Yaskawa INFORM job: OK_R2_O55(0,90)_AWOK.JBI

/JOB
//NAME OK_R2_O55(0,90)_AWOK
///FOLDERNAME X4
//POS
///NPOS 380,380,380,6,0,0
///TOOL 0
///POSTYPE PULSE
///PULSE
C00000=-116137,-64682,-98842,-22895,83957,21003
C00001=-118970,-58791,-94528,-21719,83626,20151
C00002=-128709,-21936,-78165,-7667,99802,18846
C00003=-128709,-23747,-77378,-7629,98400,18933
C00004=-129436,-40962,-90086,-7600,97096,18720
C00005=-119723,-61472,-87397,-21694,78070,20911
C00006=-121447,-61479,-87400,-20976,77655,20398
C00007=-122276,-61450,-87381,-20627,77465,20150
C00008=-121447,-61479,-87400,-20976,77655,20398
C00009=-119962,-55971,-84809,-21515,79163,20631
C00010=-119972,-52981,-83428,-21469,79803,20512
C00011=-119962,-55971,-84809,-21515,79163,20631
C00012=-118927,-58061,-86775,-21934,79541,20910
C00013=-116191,-63318,-91619,-23033,80483,21654
C00014=-116206,-56841,-96943,-22807,86586,20479
C00015=-116389,-60342,-95375,-22789,83985,20915
C00016=-116893,-39967,-83874,-22518,87009,20183
C00017=-125017,-21387,-77981,-10790,100136,18660
C00018=-125017,-23744,-76950,-10720,98321,18819
C00019=-116787,-42854,-87540,-22390,92348,19284
C00020=-121082,-61460,-87305,-21133,77696,20515
C00021=-121082,-61460,-87305,-21133,77696,20515
C00022=-122532,-61410,-87275,-20524,77362,20082
C00023=-121082,-61460,-87305,-21133,77696,20515
C00024=-120060,-56933,-85154,-21492,78877,20650
C00025=-120072,-53043,-83376,-21432,79719,20494
C00026=-120060,-56933,-85154,-21492,78877,20650
C00027=-119021,-59046,-87123,-21913,79246,20933
C00028=-116273,-64366,-91974,-23018,80167,21688
C00029=-116287,-57977,-97359,-22777,86263,20515
C00030=-114907,-63183,-96670,-23411,83739,21445
C00031=-115618,-41571,-84692,-23045,87010,20581
C00032=-116115,-23132,-74965,-22736,98208,18438
C00033=-116115,-24314,-74310,-22669,97276,18619
C00034=-115586,-41490,-86592,-22768,96199,18989
C00035=-121083,-61695,-87340,-21139,77603,20531
C00036=-121083,-61695,-87340,-21139,77603,20531
C00037=-122529,-61648,-87311,-20532,77268,20097
C00038=-121083,-61695,-87340,-21139,77603,20531
C00039=-120059,-57166,-85192,-21498,78788,20666
C00040=-120072,-53268,-83414,-21438,79633,20510
C00041=-120059,-57166,-85192,-21498,78788,20666
C00042=-119019,-59284,-87162,-21920,79155,20951
C00043=-116268,-64618,-92014,-23026,80071,21708
C00044=-116282,-58266,-97419,-22781,86162,20535
C00045=-116234,-65654,-98856,-22870,83480,21063
C00046=-117001,-30938,-83151,-22477,97538,18275
C00047=-117162,-27122,-76676,-22301,95626,18585
C00048=-117162,-28033,-76136,-22264,94882,18725
C00049=-116792,-43513,-86705,-22330,93619,19076
C00050=-121083,-61930,-87375,-21146,77510,20548
C00051=-121083,-61930,-87375,-21146,77510,20548
C00052=-122667,-61875,-87342,-20480,77145,20073
C00053=-121083,-61930,-87375,-21146,77510,20548
C00054=-120059,-57398,-85231,-21504,78698,20682
C00055=-120071,-53441,-83423,-21444,79555,20523
C00056=-120059,-57398,-85231,-21504,78698,20682
C00057=-119017,-59522,-87201,-21927,79064,20968
C00058=-116262,-64869,-92054,-23034,79975,21729
C00059=-116277,-58554,-97479,-22785,86060,20556
C00060=-116228,-66833,-98171,-22911,82531,21247
C00061=-117126,-25406,-79498,-22565,100598,17692
C00062=-117248,-21815,-74608,-22429,99491,17867
C00063=-117248,-22912,-74026,-22358,98638,18029
C00064=-116836,-40210,-86441,-22404,97572,18358
C00065=-121084,-62164,-87410,-21153,77417,20564
C00066=-121084,-62164,-87410,-21153,77417,20564
C00067=-122661,-62109,-87376,-20489,77054,20090
C00068=-121084,-62164,-87410,-21153,77417,20564
C00069=-120058,-57630,-85269,-21511,78609,20699
C00070=-120070,-53643,-83448,-21448,79472,20539
C00071=-120058,-57630,-85269,-21511,78609,20699
C00072=-119015,-59759,-87239,-21934,78973,20985
C00073=-116257,-65120,-92093,-23043,79880,21749
C00074=-116279,-54556,-99745,-22770,89251,19950
C00075=-114774,-111312,-123896,-23941,76439,22953
C00076=-117925,-58719,-95873,-21124,87917,23523
C00077=-103186,-10021,-58133,-44610,101398,29068
C00078=-123420,-23872,-71025,-15792,95845,28310
C00079=-125311,-21429,-67110,-15147,94424,27919
C00080=-120634,-65913,-76142,-32119,72760,24735
C00081=-119236,-64284,-74350,-32649,73056,25211
C00082=-125319,-21707,-67309,-15144,94403,27919
C00083=-125467,-27325,-70565,-15073,93526,27983
C00084=-125604,-31584,-72851,-15014,92748,28038
C00085=-123522,-33905,-76479,-15704,94095,28507
C00086=-123564,-36325,-78032,-15683,93810,28531
C00087=-119101,-30822,-74067,-21861,99204,35368
C00088=-119596,-32319,-75056,-21718,98940,35258
C00089=-119766,-30799,-71819,-21590,97773,35415
C00090=-121301,-29842,-70621,-21174,97189,35027
C00091=-119239,-57603,-89587,-23561,101073,42379
C00092=-120637,-57975,-90978,-23357,101328,41854
C00093=-121301,-29842,-70621,-21174,97189,35027
C00094=-121414,-33462,-72174,-21093,96316,35147
C00095=-121364,-37608,-74051,-21057,95413,35322
C00096=-118165,-36043,-78158,-22099,99263,35661
C00097=-118125,-31017,-84138,-22729,105083,34553
C00098=-120714,-60708,-105430,-21771,102512,34247
C00099=-95484,-136154,-93871,-55672,51405,46786
C00100=-114713,-99798,-82990,-41844,49051,35906
C00101=-120637,-59624,-88700,-22681,87253,37649
C00102=-119238,-59498,-87405,-23139,86931,38179
C00103=-114711,-99839,-83005,-41852,49043,35911
C00104=-114545,-102590,-83009,-42762,48062,36535
C00105=-114219,-107980,-82478,-44894,45954,37960
C00106=-111898,-109767,-89828,-42010,51787,36738
C00107=-111805,-126727,-95079,-45212,47795,38991
C00108=-66535,-95601,-84684,-52007,78764,46851
C00109=-75218,-92548,-82480,-50699,74029,44853
C00110=-81141,-84946,-78957,-49165,71925,42856
C00111=-123268,-63523,-79231,-37570,63516,21441
C00112=-124736,-66195,-80529,-37014,62443,21190
C00113=-81122,-84998,-78949,-49177,71915,42872
C00114=-79718,-88775,-78946,-49929,71393,43910
C00115=-78361,-92195,-78675,-50655,70883,44930
C00116=-68284,-113231,-96700,-52052,76723,47086
C00117=-66672,-117056,-107174,-51639,80473,45806
C00118=-77691,-86619,-95818,-48386,80174,40315
C00119=-95685,-48808,-84743,-25370,87231,35181
C00120=-95685,-48808,-84743,-25370,87231,35181
C00121=-101056,-45173,-78089,-23427,83774,34106
C00122=-102119,-43985,-76293,-23044,83049,33893
C00123=-122027,-64752,-74386,33128,72903,-25284
C00124=-120634,-66395,-76191,32602,72601,-24811
C00125=-102106,-44094,-76359,-23049,83038,33899
C00126=-101400,-49999,-79288,-23366,82078,34324
C00127=-100787,-55009,-81515,-23654,81130,34721
C00128=-99386,-53621,-81963,-24126,82412,34943
C00129=-94381,-41540,-79397,-29257,97383,37091
C00130=-94381,-42754,-78179,-29152,96177,37399
C00131=-94595,-42729,-76833,-29043,95394,37523
C00132=-96175,-42441,-75420,-28594,94264,37251
C00133=-120637,-58450,-91149,23792,101183,-41860
C00134=-122028,-58068,-89746,23994,100932,-42385
C00135=-96165,-42504,-75459,-28596,94259,37256
C00136=-95794,-45065,-76561,-28658,93810,37497
C00137=-95105,-50085,-78357,-28765,92724,38011
C00138=-93482,-48166,-78689,-29220,94287,38194
C00139=-91547,-49523,-92929,-30449,101938,36857
C00140=-111094,-45126,-96422,5689,101572,-12606
C00141=-121972,-50267,-96226,12386,99274,-20777
C00142=-120632,-57742,-90169,23117,88968,-37302
C00143=-120632,-59368,-88362,23119,87170,-37649
C00144=-119891,-47131,-80888,22873,88542,-37139
C00145=-122028,-59922,-87589,23577,86831,-38184
C00146=-120637,-60056,-88897,23120,87149,-37655
C00147=-119891,-47131,-80888,22873,88542,-37139
C00148=-120005,-53355,-83923,22914,87335,-37405
C00149=-119935,-58609,-86237,22903,86131,-37610
C00150=-123325,-57174,-87874,23990,88618,-38260
C00151=-124456,-73122,-93330,24403,84490,-39484
C00152=-120301,-77332,-95283,21145,80945,-36635
C00153=-117644,-75175,-92925,20247,79987,-35884
C00154=-120632,-66782,-80600,39533,64000,-22464
C00155=-122028,-63953,-79218,40005,65086,-22660
C00156=-117642,-75287,-92977,20248,79962,-35887
C00157=-117577,-78550,-93986,20282,78953,-36035
C00158=-117430,-84106,-95504,20358,77113,-36296
C00159=-121605,-82442,-100182,21565,81626,-36962
C00160=-121605,-75018,-107752,21416,89537,-35553
C00161=-98045,-149302,-129631,14244,61097,-31502
C00162=-124074,-173592,-119291,35973,43889,-32820
C00163=-132864,-143257,-102711,42749,53298,-34446
C00164=-130839,-124766,-99786,38797,58274,-31089
C00165=-123631,-118072,-96989,34608,55995,-27816
C00166=-123631,-118072,-96989,34608,55995,-27816
C00167=-123717,-121009,-96897,35249,54734,-28334
C00168=-124024,-127264,-96467,36865,52023,-29582
C00169=-126943,-131602,-98873,38274,52691,-30822
C00170=-128360,-153372,-105295,42598,47752,-34029
C00171=-79453,-131856,-104511,4352,44365,-9914
C00172=-78436,-115658,-92400,1620,36378,-6800
C00173=-77806,-111855,-90740,987,37302,-6435
C00174=-120634,-65728,-76133,-32106,72837,24713
C00175=-119238,-64103,-74341,-32635,73130,25188
C00176=-77806,-111855,-90740,987,37302,-6435
C00177=-76429,-114788,-90587,-338,35694,-5673
C00178=-73763,-118985,-89653,-3164,33028,-4038
C00179=-66359,-139525,-96150,-13144,27249,1592
C00180=-66359,-164100,-123806,-11486,31545,742
C00181=-70302,-83518,-108233,-11696,76370,-6987
C00182=-79254,-60990,-87055,-7574,73946,-9698
C00183=-79142,-57343,-85120,-7603,74633,-9705
C00184=-85366,-48204,-80333,1212,78686,-14938
C00185=-119241,-57353,-89541,-23570,101165,42360
C00186=-120637,-57719,-90930,-23367,101422,41835
C00187=-85366,-48204,-80333,1212,78686,-14938
C00188=-84294,-52923,-82551,739,77615,-14611
C00189=-82864,-58973,-85150,105,76099,-14163
C00190=-83777,-59837,-86544,514,76516,-14454
C00191=-81015,-69582,-89979,-723,73625,-13560
C00192=-84711,-68031,-88236,4430,73597,-17336
C00193=-120637,-59381,-88659,-22680,87345,37632
C00194=-119240,-59261,-87366,-23138,87022,38161
C00195=-84711,-68031,-88236,4430,73597,-17336
C00196=-83691,-72246,-89459,4003,72137,-17046
C00197=-83032,-75359,-90390,3727,71082,-16859
C00198=-84024,-76098,-91808,4166,71620,-17177
C00199=-84024,-66051,-103222,3998,83778,-16777
C00200=-65662,-31425,-83606,-4017,89486,-11563
C00201=-68948,-27521,-69076,-2600,82448,-12318
C00202=-64522,-19418,-61513,-8839,82863,-8015
C00203=-119239,-63197,-79148,-39462,65333,22543
C00204=-120631,-66018,-80525,-38983,64255,22343
C00205=-64522,-19418,-61513,-8839,82863,-8015
C00206=-63064,-23118,-63668,-9464,82443,-7541
C00207=-61424,-27145,-65833,-10171,81894,-6997
C00208=-62353,-28195,-68036,-9762,82596,-7338
C00209=-64122,-27053,-68918,-6328,85296,-12363
C00210=-62252,-32477,-70641,-7099,83718,-11715
C00211=-63845,-35903,-70208,-3997,79095,-11410
C00212=-122025,-64571,-74378,33114,72977,-25261
C00213=-120634,-66211,-76182,32588,72677,-24788
C00214=-63845,-35903,-70208,-3997,79095,-11410
C00215=-62658,-39020,-71374,-4529,78269,-11011
C00216=-61692,-41451,-72189,-4965,77573,-10680
C00217=-64197,-44187,-78529,-3833,79939,-11548
C00218=-64197,-33780,-85787,-3792,89732,-11844
C00219=-44689,-70929,-106175,-12114,84890,-5931
C00220=-33806,-93502,-88404,-27904,59082,13170
C00221=-58177,-75417,-81541,-6000,56276,1441
C00222=-58430,-67739,-76898,-5771,57341,1282
C00223=-120637,-58195,-91102,23802,101277,-41841
C00224=-122027,-57818,-89700,24003,101023,-42366
C00225=-58430,-67739,-76898,-5771,57341,1282
C00226=-58984,-71347,-77159,-3299,55423,-230
C00227=-57144,-74611,-77050,-4586,53771,576
C00228=-50982,-91677,-90407,-7950,54776,1850
C00229=-50982,-85567,-109418,-6960,69497,875
C00230=-54812,-62849,-98997,-4717,74482,-585
C00231=-50289,-1036,-61538,-16344,96039,-3895
C00232=-52048,7040,-42367,-12868,86243,-4159
C00233=-56434,8881,-38977,-5883,83428,-8939
C00234=-122026,-59684,-87550,23576,86921,-38166
C00235=-120637,-59813,-88856,23120,87241,-37637
C00236=-56434,8881,-38977,-5883,83428,-8939
C00237=-55375,6495,-40648,-6339,83302,-8616
C00238=-53560,2556,-43263,-7119,83025,-8054
C00239=-54077,1434,-44695,-6896,83288,-8224
C00240=-50741,-4405,-49866,-7836,84192,-7156
C00241=-51041,-4740,-48575,-7721,83208,-7185
C00242=-51232,-2335,-46154,-7645,82940,-7226
C00243=-120632,-66582,-80584,39505,64073,-22434
C00244=-122026,-63754,-79201,39978,65156,-22630
C00245=-51232,-2335,-46154,-7645,82940,-7226
C00246=-50099,-4713,-47267,-8126,82505,-6854
C00247=-49243,-6461,-48043,-8490,82167,-6570
C00248=-50339,-8396,-52000,-8013,83495,-6993
C00249=-50339,-276,-57860,-7996,91201,-7484
C00250=-32565,-26345,-77616,-15225,92076,-2559
C00251=-32565,-33689,-72287,-15210,85259,-1719
C00252=-38687,-36831,-55238,-24407,59977,6052
C00253=-39203,-33265,-53072,-24000,60287,5772
C00254=-120634,-65542,-76123,-32092,72913,24690
C00255=-119239,-63920,-74332,-32621,73204,25165
C00256=-39203,-33265,-53072,-24000,60287,5772
C00257=-37714,-35062,-52939,-25083,59795,6495
C00258=-35590,-37744,-52712,-26656,59062,7564
C00259=-26545,-57404,-66697,-31827,60841,10944
C00260=-20629,-19497,-42558,-33469,66981,11514
C00261=-27693,-14289,-39743,-29849,65249,9144
C00262=-34880,-670,-29098,-19183,60278,2827
C00263=-35092,1454,-27069,-19082,60082,2779
C00264=-119242,-57104,-89496,-23579,101256,42341
C00265=-120637,-57464,-90882,-23377,101516,41817
C00266=-35092,1454,-27069,-19082,60082,2779
C00267=-33603,-474,-27156,-20166,59534,3463
C00268=-32057,-2336,-26931,-21326,58881,4207
C00269=-32408,-6201,-31843,-20897,59764,3889
C00270=-24820,-12827,-37041,-25332,61618,6510
C00271=-24820,-941,-54339,-22867,76995,3228
C00272=-42185,7615,-42322,-13268,70874,-1244
C00273=-42932,41857,-5727,-16679,81128,-4248
C00274=-120637,-59139,-88618,-22679,87437,37614
C00275=-119242,-59024,-87327,-23137,87112,38143
C00276=-42935,41623,-5955,-16677,81147,-4251
C00277=-41455,39000,-8178,-17284,81445,-3818
C00278=-40207,36838,-9888,-17795,81632,-3440
C00279=-40859,34117,-14035,-17490,82609,-3791
C00280=-37683,30675,-15388,-18805,82352,-2733
C00281=-37683,30675,-15388,-18805,82352,-2733
C00282=-37615,32337,-12840,-18862,81691,-2611
C00283=-119240,-62997,-79129,-39436,65404,22513
C00284=-120631,-65817,-80509,-38956,64328,22314
C00285=-37615,32337,-12840,-18862,81691,-2611
C00286=-36831,30953,-13603,-19182,81626,-2349
C00287=-35920,29533,-14307,-19552,81540,-2037
C00288=-36765,31666,-24197,-19069,88162,-3353
C00289=-80819,-21628,-74687,-2656,88110,49135
C00290=-52229,28768,-25499,-44312,108635,44591
C00291=-56025,35229,-16083,-42906,105184,44544
C00292=-61493,29391,-19794,-36258,100135,45607
C00293=-62872,29148,-18454,-35815,98844,45518
C00294=-122023,-64389,-74369,33100,73050,-25238
C00295=-120634,-66025,-76173,32574,72753,-24766
C00296=-62615,28475,-19058,-35877,98962,45577
C00297=-61224,24817,-22216,-36208,99536,45909
C00298=-60367,22322,-24134,-36395,99777,46151
C00299=-59915,24005,-23707,-36577,100438,46097
C00300=-56946,22626,-23553,-38393,103359,48615
C00301=-57829,21509,-23426,-38110,102492,48585
C00302=-120637,-57938,-91054,23812,101371,-41822
C00303=-122025,-57567,-89654,24013,101115,-42346
C00304=-57829,21509,-23426,-38110,102492,48585
C00305=-56932,18945,-24988,-38222,102566,48914
C00306=-56106,16994,-26094,-38319,102642,49215
C00307=-54980,21729,-25214,-38868,104590,48938
C00308=-54302,30399,-28737,-40542,110020,47060
C00309=-40953,8747,-49252,-43839,116433,49649
C00310=-43706,2890,-35678,-39962,106692,52751
C00311=-46557,4892,-23316,-53006,96166,51821
C00312=-122025,-59445,-87511,23574,87012,-38148
C00313=-120637,-59568,-88815,23119,87334,-37619
C00314=-46557,4892,-23316,-53006,96166,51821
C00315=-45252,2504,-23846,-53101,96327,52417
C00316=-43850,228,-24056,-53173,96460,53085
C00317=-40014,1377,-25111,-53867,99354,53399
C00318=-32910,-4730,-38816,-56031,106441,52743
C00319=-47083,-38904,-60179,-52956,95987,51646
C00320=-56245,-29117,-51675,-51253,90891,49843
C00321=-59207,-29685,-49787,-50620,88366,49736
C00322=-120632,-66381,-80568,39477,64146,-22405
C00323=-122024,-63554,-79183,39951,65226,-22600
C00324=-59207,-29685,-49787,-50620,88366,49736
C00325=-57910,-32588,-50321,-50873,88309,50423
C00326=-56386,-35626,-50587,-51149,88234,51241
C00327=-48005,-36349,-53024,-52514,93554,52587
C00328=-45972,-31923,-70966,-54898,102784,48011
C00329=-62213,-2026,-48801,-50558,95689,44317
C00330=-71635,-10765,-49348,-38257,85995,47822
C00331=-73562,-12108,-48704,-37621,84358,47652
C00332=-120634,-65355,-76113,-32078,72990,24668
C00333=-119241,-63738,-74323,-32607,73278,25142
C00334=-73562,-12108,-48704,-37621,84358,47652
C00335=-72319,-16326,-51343,-38077,84425,48112
C00336=-71460,-18971,-52889,-38389,84454,48442
C00337=-69249,-19212,-54152,-39109,85879,48797
C00338=-68409,7690,-37813,-43127,101148,56069
C00339=-66304,155,-40606,-43261,100476,57243
C00340=-68124,-581,-39889,-42746,99066,57077
C00341=-119244,-56851,-89448,-23589,101349,42322
C00342=-120637,-57205,-90833,-23387,101611,41798
C00343=-68124,-581,-39889,-42746,99066,57077
C00344=-67510,-2508,-40929,-42832,99077,57331
C00345=-66648,-5140,-42298,-42942,99083,57691
C00346=-65956,-2564,-42142,-43266,100302,57463
C00347=-64160,8326,-48156,-45635,107840,54777
C00348=-82891,-1763,-56772,-40060,100398,50695
C00349=-87672,-9018,-50191,-37820,92424,51832
C00350=-88713,-8713,-49183,-37485,91645,51714
C00351=-120636,-58892,-88576,-22679,87531,37597
C00352=-119243,-58782,-87287,-23135,87203,38125
C00353=-88713,-8713,-49183,-37485,91645,51714
C00354=-87862,-13103,-52108,-37724,91615,52052
C00355=-87153,-16713,-54260,-37916,91475,52374
C00356=-86564,-15302,-54870,-38138,92586,52206
C00357=-81758,-3749,-44861,-44343,103015,58118
C00358=-82859,-4851,-44447,-43969,101921,58133
C00359=-83726,-5948,-44324,-43688,101062,58138
C00360=-119242,-62796,-79110,-39409,65475,22484
C00361=-120631,-65615,-80491,-38929,64402,22285
C00362=-83726,-5948,-44324,-43688,101062,58138
C00363=-83153,-8645,-45822,-43726,100977,58421
C00364=-82498,-11692,-47360,-43751,100817,58774
C00365=-79946,-9385,-47908,-44504,103092,58867
C00366=-79946,982,-56626,-47228,110687,55169
C00367=-67961,-35581,-83522,-49317,114444,58500
C00368=-66559,-58522,-69059,-49468,91172,57867
C00369=-76672,-55097,-64494,-49467,77742,54734
C00370=-122022,-64207,-74360,33086,73124,-25215
C00371=-120634,-65839,-76164,32560,72829,-24743
C00372=-76672,-55097,-64494,-49467,77742,54734
C00373=-75645,-58080,-64974,-49897,77474,55402
C00374=-74048,-62341,-65191,-50569,76997,56494
C00375=-72098,-59878,-66217,-50707,79300,56246
C00376=-48660,-78559,-75441,-54167,90144,62579
C00377=-24519,-71348,-75508,-48873,52324,28946
C00378=-2117,-60454,-47312,-54295,7475,4900
C00379=-2158,-60407,-47353,-53850,7490,4702
BC00000=362177,692409,1075175
BC00001=362177,692409,1075175
BC00002=362177,692409,1075175
BC00003=362177,692409,1075175
BC00004=362177,692409,1075175
BC00005=362177,692409,1075175
BC00006=362177,692409,1075175
BC00007=362177,692409,1075175
BC00008=362177,692409,1075175
BC00009=362177,692409,1075175
BC00010=362177,692409,1075175
BC00011=362177,692409,1075175
BC00012=362177,692409,1075175
BC00013=362177,692409,1075175
BC00014=362177,692409,1075175
BC00015=314570,692300,1075175
BC00016=314570,692300,1075175
BC00017=314571,692301,1075171
BC00018=314571,692301,1075171
BC00019=314570,692300,1075175
BC00020=314570,692300,1075175
BC00021=314570,692300,1075175
BC00022=314570,692300,1075175
BC00023=314570,692300,1075175
BC00024=314570,692300,1075175
BC00025=314570,692300,1075175
BC00026=314570,692300,1075175
BC00027=314570,692300,1075175
BC00028=314570,692300,1075175
BC00029=314570,692300,1075175
BC00030=266548,692394,1075175
BC00031=266548,692394,1075175
BC00032=266548,692394,1075175
BC00033=266548,692394,1075175
BC00034=266548,692394,1075175
BC00035=266548,692394,1075175
BC00036=266548,692394,1075175
BC00037=266548,692394,1075175
BC00038=266548,692394,1075175
BC00039=266548,692394,1075175
BC00040=266548,692394,1075175
BC00041=266548,692394,1075175
BC00042=266548,692394,1075175
BC00043=266548,692394,1075175
BC00044=266548,692394,1075175
BC00045=218526,692488,1075175
BC00046=218526,692488,1075175
BC00047=218526,692488,1075175
BC00048=218526,692488,1075175
BC00049=218526,692488,1075175
BC00050=218526,692488,1075175
BC00051=218526,692488,1075175
BC00052=218526,692488,1075175
BC00053=218526,692488,1075175
BC00054=218526,692488,1075175
BC00055=218526,692488,1075175
BC00056=218526,692488,1075175
BC00057=218526,692488,1075175
BC00058=218526,692488,1075175
BC00059=218526,692488,1075175
BC00060=170743,692582,1075175
BC00061=170743,692582,1075175
BC00062=170743,692582,1075175
BC00063=170743,692582,1075175
BC00064=170743,692582,1075175
BC00065=170743,692582,1075175
BC00066=170743,692582,1075175
BC00067=170743,692582,1075175
BC00068=170743,692582,1075175
BC00069=170743,692582,1075175
BC00070=170743,692582,1075175
BC00071=170743,692582,1075175
BC00072=170743,692582,1075175
BC00073=170743,692582,1075175
BC00074=170743,692582,1075175
BC00075=170743,673726,1075175
BC00076=170861,676324,1075173
BC00077=170861,676324,1075173
BC00078=171122,682063,1075169
BC00079=171122,682063,1075169
BC00080=184393,664970,1075175
BC00081=184393,664970,1075175
BC00082=171122,682063,1075169
BC00083=171122,682063,1075169
BC00084=171122,682063,1075169
BC00085=171122,682063,1075169
BC00086=171122,682063,1075169
BC00087=171122,682063,1075169
BC00088=171122,682063,1075169
BC00089=171122,682063,1075169
BC00090=171122,682063,1075169
BC00091=173178,720507,1075175
BC00092=173178,720507,1075175
BC00093=171122,682063,1075169
BC00094=171122,682063,1075169
BC00095=171122,682063,1075169
BC00096=171122,682063,1075169
BC00097=171122,682063,1075169
BC00098=171122,682063,1075169
BC00099=171122,682063,1075169
BC00100=171122,682063,1075169
BC00101=173051,704467,1075175
BC00102=173051,704467,1075175
BC00103=171122,682063,1075169
BC00104=171122,682063,1075169
BC00105=171122,682063,1075169
BC00106=171498,685555,1075169
BC00107=171498,685555,1075169
BC00108=171498,685555,1075169
BC00109=171498,685555,1075169
BC00110=171498,685555,1075169
BC00111=196106,690466,1075175
BC00112=196106,690466,1075175
BC00113=171498,685555,1075169
BC00114=171498,685555,1075169
BC00115=171498,685555,1075169
BC00116=171498,685555,1075169
BC00117=171498,685555,1075169
BC00118=171498,685555,1075169
BC00119=171731,685521,1075169
BC00120=171731,685521,1075169
BC00121=171731,685521,1075169
BC00122=171731,685521,1075169
BC00123=58729,665797,1075175
BC00124=58729,665797,1075175
BC00125=171731,685521,1075169
BC00126=171731,685521,1075169
BC00127=171731,685521,1075169
BC00128=171731,685521,1075169
BC00129=171731,685521,1075169
BC00130=171731,685521,1075169
BC00131=171731,685521,1075169
BC00132=171731,685521,1075169
BC00133=70497,721413,1075175
BC00134=70497,721413,1075175
BC00135=171731,685521,1075169
BC00136=171731,685521,1075169
BC00137=171731,685521,1075169
BC00138=171731,685521,1075169
BC00139=171731,685521,1075169
BC00140=98396,696294,1075173
BC00141=90128,697509,1075173
BC00142=62613,701551,1075175
BC00143=68182,704259,1075175
BC00144=69760,705026,1075175
BC00145=70409,705342,1075175
BC00146=70409,705342,1075175
BC00147=69760,705026,1075175
BC00148=69760,705026,1075175
BC00149=69760,705026,1075175
BC00150=69760,705026,1075175
BC00151=69760,705026,1075175
BC00152=69760,705026,1075175
BC00153=69760,705026,1075175
BC00154=53891,691077,1075175
BC00155=53891,691077,1075175
BC00156=69760,705026,1075175
BC00157=69760,705026,1075175
BC00158=69760,705026,1075175
BC00159=69760,705026,1075175
BC00160=69760,705026,1075175
BC00161=69760,705026,1075175
BC00162=69760,705026,1075175
BC00163=69760,705026,1075175
BC00164=69760,705026,1075175
BC00165=69760,705026,1075175
BC00166=69760,705026,1075175
BC00167=69760,705026,1075175
BC00168=69760,705026,1075175
BC00169=69760,705026,1075175
BC00170=69760,705026,1075175
BC00171=69760,705026,1075175
BC00172=69760,705026,1075175
BC00173=69760,705026,1075175
BC00174=232176,664876,1075175
BC00175=232176,664876,1075175
BC00176=69760,705026,1075175
BC00177=69760,705026,1075175
BC00178=69760,705026,1075171
BC00179=69760,705026,1075171
BC00180=69760,705026,1075171
BC00181=69760,705026,1075171
BC00182=69760,705026,1075171
BC00183=69760,705026,1075171
BC00184=69760,705026,1075171
BC00185=220961,720413,1075175
BC00186=220961,720413,1075175
BC00187=69760,705026,1075171
BC00188=69760,705026,1075171
BC00189=69760,705026,1075171
BC00190=69760,705026,1075171
BC00191=69760,705026,1075171
BC00192=69760,705026,1075171
BC00193=220834,704373,1075175
BC00194=220834,704373,1075175
BC00195=69760,705026,1075171
BC00196=69760,705026,1075171
BC00197=69760,705026,1075171
BC00198=69760,705026,1075171
BC00199=69760,705026,1075171
BC00200=69760,705026,1075171
BC00201=69760,705026,1075171
BC00202=69760,705026,1075171
BC00203=236979,690198,1075175
BC00204=236979,690198,1075175
BC00205=69760,705026,1075171
BC00206=69760,705026,1075171
BC00207=69760,705026,1075171
BC00208=69760,705026,1075171
BC00209=69760,705026,1075171
BC00210=69760,705026,1075171
BC00211=69760,705026,1075171
BC00212=106512,665703,1075175
BC00213=106512,665703,1075175
BC00214=69760,705026,1075171
BC00215=69760,705026,1075171
BC00216=69760,705026,1075171
BC00217=69760,705026,1075171
BC00218=69760,705026,1075171
BC00219=69760,705026,1075171
BC00220=69760,705026,1075171
BC00221=70001,705106,1075155
BC00222=70001,705106,1075155
BC00223=118281,721319,1075175
BC00224=118281,721319,1075175
BC00225=70001,705106,1075155
BC00226=70001,705106,1075161
BC00227=70001,705106,1075165
BC00228=72274,705262,1075165
BC00229=72274,705262,1075165
BC00230=72274,705262,1075165
BC00231=72274,705262,1075165
BC00232=72274,705262,1075165
BC00233=72274,705262,1075165
BC00234=118193,705249,1075175
BC00235=118193,705249,1075175
BC00236=72274,705262,1075165
BC00237=72274,705262,1075165
BC00238=72274,705262,1075165
BC00239=72274,705262,1075165
BC00240=72274,705262,1075165
BC00241=72274,705262,1075165
BC00242=72274,705262,1075165
BC00243=101675,690983,1075175
BC00244=101675,690983,1075175
BC00245=72274,705262,1075165
BC00246=72274,705262,1075165
BC00247=72274,705262,1075165
BC00248=72274,705262,1075165
BC00249=72274,705262,1075165
BC00250=72274,705262,1075165
BC00251=72274,705262,1075165
BC00252=72274,705262,1075165
BC00253=72274,705262,1075165
BC00254=280198,664783,1075175
BC00255=280198,664783,1075175
BC00256=72274,705262,1075165
BC00257=72274,705262,1075165
BC00258=72274,705262,1075165
BC00259=72274,705262,1075165
BC00260=72274,705262,1075165
BC00261=72274,705262,1075165
BC00262=72274,705262,1075165
BC00263=72274,705262,1075165
BC00264=268505,720320,1075175
BC00265=268505,720320,1075175
BC00266=72274,705262,1075165
BC00267=72274,705262,1075165
BC00268=72274,705262,1075165
BC00269=72274,705262,1075165
BC00270=72274,705262,1075165
BC00271=72274,705262,1075165
BC00272=72274,705262,1075165
BC00273=72274,705261,1075162
BC00274=268378,704280,1075175
BC00275=268378,704280,1075175
BC00276=72274,705261,1075162
BC00277=72274,705262,1075165
BC00278=72274,705262,1075165
BC00279=72274,705262,1075165
BC00280=72274,705262,1075165
BC00281=72274,705262,1075165
BC00282=72274,705262,1075165
BC00283=285001,690104,1075175
BC00284=285001,690104,1075175
BC00285=72274,705262,1075165
BC00286=72274,705262,1075165
BC00287=72274,705262,1075165
BC00288=71257,705262,1075165
BC00289=200486,668518,1075165
BC00290=200486,668518,1075165
BC00291=200486,668518,1075165
BC00292=200486,668518,1075165
BC00293=200486,668518,1075165
BC00294=154534,665609,1075175
BC00295=154534,665609,1075175
BC00296=200486,668518,1075162
BC00297=200486,668518,1075162
BC00298=200486,668518,1075162
BC00299=200486,668518,1075162
BC00300=200486,668518,1075162
BC00301=200487,668518,1075159
BC00302=166303,721225,1075175
BC00303=166303,721225,1075175
BC00304=200487,668518,1075159
BC00305=200487,668518,1075159
BC00306=200487,668518,1075159
BC00307=200487,668518,1075159
BC00308=200487,668518,1075159
BC00309=200487,668518,1075159
BC00310=200487,668518,1075159
BC00311=200487,668518,1075159
BC00312=166215,705155,1075175
BC00313=166215,705155,1075175
BC00314=200487,668518,1075159
BC00315=200487,668518,1075159
BC00316=200487,668518,1075155
BC00317=200487,668518,1075152
BC00318=200487,668518,1075152
BC00319=200487,668518,1075152
BC00320=200487,668518,1075152
BC00321=200487,668518,1075152
BC00322=149697,690889,1075175
BC00323=149697,690889,1075175
BC00324=200487,668518,1075152
BC00325=200487,668518,1075152
BC00326=200487,668518,1075152
BC00327=200487,668518,1075152
BC00328=200487,668518,1075152
BC00329=200487,668518,1075152
BC00330=200487,668518,1075152
BC00331=200487,668518,1075152
BC00332=328220,664689,1075175
BC00333=328220,664689,1075175
BC00334=200487,668518,1075152
BC00335=200487,668518,1075152
BC00336=200487,668518,1075152
BC00337=200487,668518,1075152
BC00338=200487,668518,1075152
BC00339=200487,668518,1075152
BC00340=200487,668518,1075152
BC00341=317005,720225,1075175
BC00342=317005,720225,1075175
BC00343=200487,668518,1075152
BC00344=200487,668518,1075152
BC00345=200487,668518,1075152
BC00346=200487,668518,1075152
BC00347=200487,668518,1075152
BC00348=200487,668518,1075152
BC00349=200487,668518,1075152
BC00350=200487,668518,1075152
BC00351=316878,704185,1075175
BC00352=316878,704185,1075175
BC00353=200487,668518,1075152
BC00354=200487,668518,1075152
BC00355=200487,668518,1075152
BC00356=200487,668518,1075152
BC00357=200487,668518,1075152
BC00358=200487,668518,1075152
BC00359=200487,668518,1075152
BC00360=333023,690010,1075175
BC00361=333023,690010,1075175
BC00362=200487,668518,1075152
BC00363=200487,668518,1075152
BC00364=200487,668518,1075152
BC00365=200487,668518,1075152
BC00366=200487,668518,1075152
BC00367=200487,668518,1075152
BC00368=200487,668518,1075152
BC00369=200487,668518,1075152
BC00370=202556,665515,1075175
BC00371=202556,665515,1075175
BC00372=200487,668518,1075152
BC00373=200487,668518,1075152
BC00374=200487,668518,1075152
BC00375=200487,668518,1075152
BC00376=200487,668518,1075152
BC00377=200488,668518,1075150
BC00378=200488,668518,1075149
BC00379=193993,668519,1075142
EC00000=0,556475
EC00001=0,556475
EC00002=0,556475
EC00003=0,556475
EC00004=0,556475
EC00005=0,556475
EC00006=0,556475
EC00007=0,556475
EC00008=0,556475
EC00009=0,556475
EC00010=0,556475
EC00011=0,556475
EC00012=0,556475
EC00013=0,556475
EC00014=0,556475
EC00015=0,556475
EC00016=0,556475
EC00017=1,556475
EC00018=1,556475
EC00019=0,556475
EC00020=0,556475
EC00021=0,556475
EC00022=0,556475
EC00023=0,556475
EC00024=0,556475
EC00025=0,556475
EC00026=0,556475
EC00027=0,556475
EC00028=0,556475
EC00029=0,556475
EC00030=0,556475
EC00031=0,556475
EC00032=0,556475
EC00033=0,556475
EC00034=0,556475
EC00035=0,556475
EC00036=0,556475
EC00037=0,556475
EC00038=0,556475
EC00039=0,556475
EC00040=0,556475
EC00041=0,556475
EC00042=0,556475
EC00043=0,556475
EC00044=0,556475
EC00045=0,556475
EC00046=0,556475
EC00047=0,556475
EC00048=0,556475
EC00049=0,556475
EC00050=0,556475
EC00051=0,556475
EC00052=0,556475
EC00053=0,556475
EC00054=0,556475
EC00055=0,556475
EC00056=0,556475
EC00057=0,556475
EC00058=0,556475
EC00059=0,556475
EC00060=0,556475
EC00061=0,556475
EC00062=0,556475
EC00063=0,556475
EC00064=0,556475
EC00065=0,556475
EC00066=0,556475
EC00067=0,556475
EC00068=0,556475
EC00069=0,556475
EC00070=0,556475
EC00071=0,556475
EC00072=0,556475
EC00073=0,556475
EC00074=0,556475
EC00075=0,556475
EC00076=0,556475
EC00077=0,556475
EC00078=1,556474
EC00079=1,556474
EC00080=0,556475
EC00081=0,556475
EC00082=1,556474
EC00083=1,556474
EC00084=1,556474
EC00085=1,556474
EC00086=1,556474
EC00087=1,556474
EC00088=1,556474
EC00089=1,556474
EC00090=1,556474
EC00091=0,556475
EC00092=0,556475
EC00093=1,556474
EC00094=1,556474
EC00095=1,556474
EC00096=1,556474
EC00097=1,556474
EC00098=1,556474
EC00099=1,556474
EC00100=1,556474
EC00101=0,556475
EC00102=0,556475
EC00103=1,556474
EC00104=1,556474
EC00105=1,556474
EC00106=1,556474
EC00107=1,556474
EC00108=1,556474
EC00109=1,556474
EC00110=1,556474
EC00111=0,556475
EC00112=0,556475
EC00113=1,556474
EC00114=1,556474
EC00115=1,556474
EC00116=1,556474
EC00117=1,556474
EC00118=1,556474
EC00119=1,556474
EC00120=1,556474
EC00121=1,556474
EC00122=1,556474
EC00123=0,556475
EC00124=0,556475
EC00125=1,556474
EC00126=1,556474
EC00127=1,556474
EC00128=1,556474
EC00129=1,556474
EC00130=1,556474
EC00131=1,556474
EC00132=1,556474
EC00133=0,556475
EC00134=0,556475
EC00135=1,556474
EC00136=1,556474
EC00137=1,556474
EC00138=1,556474
EC00139=1,556474
EC00140=0,556475
EC00141=0,556475
EC00142=0,556475
EC00143=0,556475
EC00144=0,556475
EC00145=0,556475
EC00146=0,556475
EC00147=0,556475
EC00148=0,556475
EC00149=0,556475
EC00150=0,556475
EC00151=0,556475
EC00152=0,556475
EC00153=0,556475
EC00154=0,556475
EC00155=0,556475
EC00156=0,556475
EC00157=0,556475
EC00158=0,556475
EC00159=0,556475
EC00160=0,556475
EC00161=0,556475
EC00162=0,556475
EC00163=0,556475
EC00164=0,556475
EC00165=0,556475
EC00166=0,556475
EC00167=0,556475
EC00168=0,556475
EC00169=0,556475
EC00170=0,556475
EC00171=0,556475
EC00172=0,556475
EC00173=0,556475
EC00174=0,556475
EC00175=0,556475
EC00176=0,556475
EC00177=0,556475
EC00178=0,556475
EC00179=0,556475
EC00180=0,556475
EC00181=0,556475
EC00182=0,556475
EC00183=0,556475
EC00184=0,556475
EC00185=0,556475
EC00186=0,556475
EC00187=0,556475
EC00188=0,556475
EC00189=0,556475
EC00190=0,556475
EC00191=0,556475
EC00192=0,556475
EC00193=0,556475
EC00194=0,556475
EC00195=0,556475
EC00196=0,556475
EC00197=0,556475
EC00198=0,556475
EC00199=0,556475
EC00200=0,556475
EC00201=0,556475
EC00202=0,556475
EC00203=0,556475
EC00204=0,556475
EC00205=0,556475
EC00206=0,556475
EC00207=0,556475
EC00208=0,556475
EC00209=0,556475
EC00210=0,556475
EC00211=0,556475
EC00212=0,556475
EC00213=0,556475
EC00214=0,556475
EC00215=0,556475
EC00216=0,556475
EC00217=0,556475
EC00218=0,556475
EC00219=0,556475
EC00220=0,556475
EC00221=3,556475
EC00222=3,556475
EC00223=0,556475
EC00224=0,556475
EC00225=3,556475
EC00226=2,556475
EC00227=1,556475
EC00228=1,556475
EC00229=1,556475
EC00230=1,556475
EC00231=1,556475
EC00232=1,556475
EC00233=1,556475
EC00234=0,556475
EC00235=0,556475
EC00236=1,556475
EC00237=1,556475
EC00238=1,556475
EC00239=1,556475
EC00240=1,556475
EC00241=1,556475
EC00242=1,556475
EC00243=0,556475
EC00244=0,556475
EC00245=1,556475
EC00246=1,556475
EC00247=1,556475
EC00248=1,556475
EC00249=1,556475
EC00250=1,556475
EC00251=1,556475
EC00252=1,556475
EC00253=1,556475
EC00254=0,556475
EC00255=0,556475
EC00256=1,556475
EC00257=1,556475
EC00258=1,556475
EC00259=1,556475
EC00260=1,556475
EC00261=1,556475
EC00262=1,556475
EC00263=1,556475
EC00264=0,556475
EC00265=0,556475
EC00266=1,556475
EC00267=1,556475
EC00268=1,556475
EC00269=1,556475
EC00270=1,556475
EC00271=1,556475
EC00272=1,556475
EC00273=1,556474
EC00274=0,556475
EC00275=0,556475
EC00276=1,556474
EC00277=1,556475
EC00278=1,556475
EC00279=1,556475
EC00280=1,556475
EC00281=1,556475
EC00282=1,556475
EC00283=0,556475
EC00284=0,556475
EC00285=1,556475
EC00286=1,556475
EC00287=1,556475
EC00288=1,556475
EC00289=1,556475
EC00290=1,556475
EC00291=1,556475
EC00292=1,556475
EC00293=1,556475
EC00294=0,556475
EC00295=0,556475
EC00296=1,556475
EC00297=1,556475
EC00298=1,556475
EC00299=1,556475
EC00300=1,556475
EC00301=2,556475
EC00302=0,556475
EC00303=0,556475
EC00304=2,556475
EC00305=2,556475
EC00306=2,556475
EC00307=2,556475
EC00308=2,556475
EC00309=2,556475
EC00310=2,556475
EC00311=2,556475
EC00312=0,556475
EC00313=0,556475
EC00314=2,556475
EC00315=2,556475
EC00316=2,556475
EC00317=3,556474
EC00318=3,556474
EC00319=3,556474
EC00320=3,556474
EC00321=3,556474
EC00322=0,556475
EC00323=0,556475
EC00324=3,556474
EC00325=3,556474
EC00326=3,556474
EC00327=3,556474
EC00328=3,556474
EC00329=3,556474
EC00330=3,556474
EC00331=3,556474
EC00332=0,556475
EC00333=0,556475
EC00334=3,556474
EC00335=3,556474
EC00336=3,556474
EC00337=3,556474
EC00338=3,556474
EC00339=3,556474
EC00340=3,556474
EC00341=0,556475
EC00342=0,556475
EC00343=3,556474
EC00344=3,556474
EC00345=3,556474
EC00346=3,556474
EC00347=3,556474
EC00348=3,556474
EC00349=3,556474
EC00350=3,556474
EC00351=0,556475
EC00352=0,556475
EC00353=3,556474
EC00354=3,556474
EC00355=3,556474
EC00356=3,556474
EC00357=3,556474
EC00358=3,556474
EC00359=3,556474
EC00360=0,556475
EC00361=0,556475
EC00362=3,556474
EC00363=3,556474
EC00364=3,556474
EC00365=3,556474
EC00366=3,556474
EC00367=3,556474
EC00368=3,556474
EC00369=3,556474
EC00370=0,556475
EC00371=0,556475
EC00372=3,556474
EC00373=3,556474
EC00374=3,556474
EC00375=3,556474
EC00376=3,556474
EC00377=4,556474
EC00378=4,556474
EC00379=5,556474
///POSTYPE BASE
///RECTAN
///RCONF 0,0,0,0,0,0,0,0,0,0,0,0,0,0,0,0,0,0,0,0,0,0,0,0
P00006=0.222,-3.123,-1.508,0.0000,0.0000,0.0000
P00031=1.853,-0.001,-1.549,0.0000,0.0000,0.0000
P00032=1.957,0.503,-7.217,0.0000,0.0000,0.0000
///RCONF 0,0,0,0,1,0,0,0,0,0,0,0,0,0,0,0,0,0,0,0,0,0,0,0
P00033=-0.123,0.612,-5.012,0.0000,0.0000,0.0000
///RCONF 0,0,0,0,0,0,0,0,0,0,0,0,0,0,0,0,0,0,0,0,0,0,0,0
P00034=-0.304,0.773,-2.693,0.0000,0.0000,0.0000
P00035=2.817,0.591,-1.622,0.0000,0.0000,0.0000
//INST
///DATE 2024/01/03 14:30
///ATTR SC,RW
///GROUP1 RB1,BS1
///GROUP2 ST1
NOP
'OK_r2_O55(0,90)
'Path S1236
SFTOF3D
MOVJ C00000 BC00000 VJ=100.00  +MOVJ EC00000 VJ=100.00
MOVL C00001 BC00001 V=400.0  +MOVJ EC00001 VJ=100.00
SMOVL C00002 BC00002 V=60.0  +MOVJ EC00002
SREFP 3 C00003 BC00003  +REFP EC00003
CALL JOB:SEARCH-R1-S13D
SET P031 P006
SFTON3D P031
SMOVL C00004 BC00004 V=60.0  +MOVJ EC00004
SMOVL C00005 BC00005 V=60.0  +MOVJ EC00005
SMOVL C00006 BC00006 V=60.0  +MOVJ EC00006
SREFP 3 C00007 BC00007  +REFP EC00007
CALL JOB:SEARCH-R1-S13D
SET P031 P006
SFTON3D P031
SMOVL C00008 BC00008 V=60.0  +MOVJ EC00008
SMOVL C00009 BC00009 V=60.0  +MOVJ EC00009
SREFP 3 C00010 BC00010  +REFP EC00010
CALL JOB:SEARCH-R1-S13D
SET P031 P006
SFTON3D P031
SMOVL C00011 BC00011 V=60.0  +MOVJ EC00011
MOVL C00012 BC00012 V=400.0  +MOVJ EC00012 VJ=100.00
MOVL C00013 BC00013 V=1000.0  +MOVJ EC00013 VJ=100.00
MOVL C00014 BC00014 V=1000.0  +MOVJ EC00014 VJ=100.00
'Path S1237
SFTOF3D
MOVJ C00015 BC00015 VJ=100.00  +MOVJ EC00015 VJ=100.00
MOVL C00016 BC00016 V=400.0  +MOVJ EC00016 VJ=100.00
SMOVL C00017 BC00017 V=60.0  +MOVJ EC00017
SREFP 3 C00018 BC00018  +REFP EC00018
CALL JOB:SEARCH-R1-S13D
SET P032 P006
SFTON3D P032
SMOVL C00019 BC00019 V=60.0  +MOVJ EC00019
SMOVL C00020 BC00020 V=60.0  +MOVJ EC00020
SMOVL C00021 BC00021 V=60.0  +MOVJ EC00021
SREFP 3 C00022 BC00022  +REFP EC00022
CALL JOB:SEARCH-R1-S13D
SET P032 P006
SFTON3D P032
SMOVL C00023 BC00023 V=60.0  +MOVJ EC00023
SMOVL C00024 BC00024 V=60.0  +MOVJ EC00024
SREFP 3 C00025 BC00025  +REFP EC00025
CALL JOB:SEARCH-R1-S13D
SET P032 P006
SFTON3D P032
SMOVL C00026 BC00026 V=60.0  +MOVJ EC00026
MOVL C00027 BC00027 V=400.0  +MOVJ EC00027 VJ=100.00
MOVL C00028 BC00028 V=1000.0  +MOVJ EC00028 VJ=100.00
MOVL C00029 BC00029 V=1000.0  +MOVJ EC00029 VJ=100.00
'Path S1238
SFTOF3D
MOVJ C00030 BC00030 VJ=100.00  +MOVJ EC00030 VJ=100.00
MOVL C00031 BC00031 V=400.0  +MOVJ EC00031 VJ=100.00
SMOVL C00032 BC00032 V=60.0  +MOVJ EC00032
SREFP 3 C00033 BC00033  +REFP EC00033
CALL JOB:SEARCH-R1-S13D
SET P033 P006
SFTON3D P033
SMOVL C00034 BC00034 V=60.0  +MOVJ EC00034
SMOVL C00035 BC00035 V=60.0  +MOVJ EC00035
SMOVL C00036 BC00036 V=60.0  +MOVJ EC00036
SREFP 3 C00037 BC00037  +REFP EC00037
CALL JOB:SEARCH-R1-S13D
SET P033 P006
SFTON3D P033
SMOVL C00038 BC00038 V=60.0  +MOVJ EC00038
SMOVL C00039 BC00039 V=60.0  +MOVJ EC00039
SREFP 3 C00040 BC00040  +REFP EC00040
CALL JOB:SEARCH-R1-S13D
SET P033 P006
SFTON3D P033
SMOVL C00041 BC00041 V=60.0  +MOVJ EC00041
MOVL C00042 BC00042 V=400.0  +MOVJ EC00042 VJ=100.00
MOVL C00043 BC00043 V=1000.0  +MOVJ EC00043 VJ=100.00
MOVL C00044 BC00044 V=1000.0  +MOVJ EC00044 VJ=100.00
'Path S1239
SFTOF3D
MOVJ C00045 BC00045 VJ=100.00  +MOVJ EC00045 VJ=100.00
MOVL C00046 BC00046 V=400.0  +MOVJ EC00046 VJ=100.00
SMOVL C00047 BC00047 V=60.0  +MOVJ EC00047
SREFP 3 C00048 BC00048  +REFP EC00048
CALL JOB:SEARCH-R1-S13D
SET P034 P006
SFTON3D P034
SMOVL C00049 BC00049 V=60.0  +MOVJ EC00049
SMOVL C00050 BC00050 V=60.0  +MOVJ EC00050
SMOVL C00051 BC00051 V=60.0  +MOVJ EC00051
SREFP 3 C00052 BC00052  +REFP EC00052
CALL JOB:SEARCH-R1-S13D
SET P034 P006
SFTON3D P034
SMOVL C00053 BC00053 V=60.0  +MOVJ EC00053
SMOVL C00054 BC00054 V=60.0  +MOVJ EC00054
SREFP 3 C00055 BC00055  +REFP EC00055
CALL JOB:SEARCH-R1-S13D
SET P034 P006
SFTON3D P034
SMOVL C00056 BC00056 V=60.0  +MOVJ EC00056
MOVL C00057 BC00057 V=400.0  +MOVJ EC00057 VJ=100.00
MOVL C00058 BC00058 V=1000.0  +MOVJ EC00058 VJ=100.00
MOVL C00059 BC00059 V=1000.0  +MOVJ EC00059 VJ=100.00
'Path S1194
SFTOF3D
MOVJ C00060 BC00060 VJ=100.00  +MOVJ EC00060 VJ=100.00
MOVL C00061 BC00061 V=400.0  +MOVJ EC00061 VJ=100.00
SMOVL C00062 BC00062 V=60.0  +MOVJ EC00062
SREFP 3 C00063 BC00063  +REFP EC00063
CALL JOB:SEARCH-R1-S13D
SET P035 P006
SFTON3D P035
SMOVL C00064 BC00064 V=60.0  +MOVJ EC00064
SMOVL C00065 BC00065 V=60.0  +MOVJ EC00065
SMOVL C00066 BC00066 V=60.0  +MOVJ EC00066
SREFP 3 C00067 BC00067  +REFP EC00067
CALL JOB:SEARCH-R1-S13D
SET P035 P006
SFTON3D P035
SMOVL C00068 BC00068 V=60.0  +MOVJ EC00068
SMOVL C00069 BC00069 V=60.0  +MOVJ EC00069
SREFP 3 C00070 BC00070  +REFP EC00070
CALL JOB:SEARCH-R1-S13D
SET P035 P006
SFTON3D P035
SMOVL C00071 BC00071 V=60.0  +MOVJ EC00071
MOVL C00072 BC00072 V=400.0  +MOVJ EC00072 VJ=100.00
MOVL C00073 BC00073 V=1000.0  +MOVJ EC00073 VJ=100.00
MOVL C00074 BC00074 V=1000.0  +MOVJ EC00074 VJ=100.00
MOVJ C00075 BC00075 VJ=100.00  +MOVJ EC00075 VJ=100.00
'
SFTOF3D
'Path W1103
SFTOF3D
SFTON3D P035
MOVJ C00076 BC00076 VJ=100.00  +MOVJ EC00076 VJ=100.00
'COMMENT
'COMMENT
SMOVL C00077 BC00077 V=60.0  +MOVJ EC00077
'COMMENT
'COMMENT
SMOVL C00078 BC00078 V=400.0  +MOVJ EC00078
SMOVL C00079 BC00079 V=100.0 PL=0  +MOVJ EC00079
SREFP 1 C00080 BC00080  +REFP EC00080
SREFP 2 C00081 BC00081  +REFP EC00081
MACRO1 MJ#(0) ARGF0
ARCON
SMOVC C00082 BC00082 V=11.0  +MOVJ EC00082
SMOVC C00083 BC00083 V=11.0  +MOVJ EC00083
SMOVC C00084 BC00084 V=11.0  +MOVJ EC00084
ARCOF
SMOVL C00085 BC00085 V=400.0  +MOVJ EC00085
SMOVL C00086 BC00086 V=1000.0  +MOVJ EC00086
SFTOF3D
MOVJ C00087 BC00087 VJ=100.00  +MOVJ EC00087 VJ=100.00
'Path W1104
SFTOF3D
SFTON3D P035
MOVJ C00088 BC00088 VJ=100.00  +MOVJ EC00088 VJ=100.00
SMOVL C00089 BC00089 V=400.0  +MOVJ EC00089
SMOVL C00090 BC00090 V=100.0 PL=0  +MOVJ EC00090
SREFP 1 C00091 BC00091  +REFP EC00091
SREFP 2 C00092 BC00092  +REFP EC00092
MACRO1 MJ#(0) ARGF0
ARCON
SMOVC C00093 BC00093 V=11.0  +MOVJ EC00093
SMOVC C00094 BC00094 V=11.0  +MOVJ EC00094
SMOVC C00095 BC00095 V=11.0  +MOVJ EC00095
ARCOF
SMOVL C00096 BC00096 V=400.0  +MOVJ EC00096
SMOVL C00097 BC00097 V=1000.0  +MOVJ EC00097
SFTOF3D
'Path W1105
SFTOF3D
SFTON3D P035
MOVJ C00098 BC00098 VJ=100.00  +MOVJ EC00098 VJ=100.00
SMOVL C00099 BC00099 V=400.0  +MOVJ EC00099
SMOVL C00100 BC00100 V=100.0 PL=0  +MOVJ EC00100
SREFP 1 C00101 BC00101  +REFP EC00101
SREFP 2 C00102 BC00102  +REFP EC00102
MACRO1 MJ#(0) ARGF0
ARCON
SMOVC C00103 BC00103 V=11.0  +MOVJ EC00103
SMOVC C00104 BC00104 V=11.0  +MOVJ EC00104
SMOVC C00105 BC00105 V=11.0  +MOVJ EC00105
ARCOF
SMOVL C00106 BC00106 V=400.0  +MOVJ EC00106
SMOVL C00107 BC00107 V=1000.0  +MOVJ EC00107
SFTOF3D
'Path W1137
SFTOF3D
SFTON3D P034
MOVJ C00108 BC00108 VJ=100.00  +MOVJ EC00108 VJ=100.00
SMOVL C00109 BC00109 V=400.0  +MOVJ EC00109
SMOVL C00110 BC00110 V=100.0 PL=0  +MOVJ EC00110
SREFP 1 C00111 BC00111  +REFP EC00111
SREFP 2 C00112 BC00112  +REFP EC00112
MACRO1 MJ#(0) ARGF0
ARCON
SMOVC C00113 BC00113 V=11.0  +MOVJ EC00113
SMOVC C00114 BC00114 V=11.0  +MOVJ EC00114
SMOVC C00115 BC00115 V=11.0  +MOVJ EC00115
ARCOF
SMOVL C00116 BC00116 V=400.0  +MOVJ EC00116
SMOVL C00117 BC00117 V=1000.0  +MOVJ EC00117
SMOVL C00118 BC00118 V=1000.0  +MOVJ EC00118
SFTOF3D
MOVJ C00119 BC00119 VJ=100.00  +MOVJ EC00119 VJ=100.00
'
'Path W1577
SFTOF3D
SFTON3D P034
MOVJ C00120 BC00120 VJ=100.00  +MOVJ EC00120 VJ=100.00
SMOVL C00121 BC00121 V=400.0  +MOVJ EC00121
SMOVL C00122 BC00122 V=100.0 PL=0  +MOVJ EC00122
SREFP 1 C00123 BC00123  +REFP EC00123
SREFP 2 C00124 BC00124  +REFP EC00124
MACRO1 MJ#(0) ARGF0
ARCON
SMOVC C00125 BC00125 V=11.0  +MOVJ EC00125
SMOVC C00126 BC00126 V=11.0  +MOVJ EC00126
SMOVC C00127 BC00127 V=11.0  +MOVJ EC00127
ARCOF
SMOVL C00128 BC00128 V=400.0  +MOVJ EC00128
SFTOF3D
MOVJ C00129 BC00129 VJ=100.00  +MOVJ EC00129 VJ=100.00
'Path W1578
SFTOF3D
SFTON3D P034
MOVJ C00130 BC00130 VJ=100.00  +MOVJ EC00130 VJ=100.00
SMOVL C00131 BC00131 V=400.0  +MOVJ EC00131
SMOVL C00132 BC00132 V=100.0 PL=0  +MOVJ EC00132
SREFP 1 C00133 BC00133  +REFP EC00133
SREFP 2 C00134 BC00134  +REFP EC00134
MACRO1 MJ#(0) ARGF0
ARCON
SMOVC C00135 BC00135 V=11.0  +MOVJ EC00135
SMOVC C00136 BC00136 V=11.0  +MOVJ EC00136
SMOVC C00137 BC00137 V=11.0  +MOVJ EC00137
ARCOF
SMOVL C00138 BC00138 V=400.0  +MOVJ EC00138
SMOVL C00139 BC00139 V=1000.0  +MOVJ EC00139
SFTOF3D
'Path W1579
SFTOF3D
SFTON3D P035
MOVJ C00140 BC00140 VJ=50.00  +MOVJ EC00140 VJ=50.00
MOVJ C00141 BC00141 VJ=50.00  +MOVJ EC00141 VJ=50.00
MOVJ C00142 BC00142 VJ=100.00  +MOVJ EC00142 VJ=100.00
SMOVL C00143 BC00143 V=400.0  +MOVJ EC00143
SMOVL C00144 BC00144 V=100.0 PL=0  +MOVJ EC00144
SREFP 1 C00145 BC00145  +REFP EC00145
SREFP 2 C00146 BC00146  +REFP EC00146
MACRO1 MJ#(0) ARGF0
ARCON
SMOVC C00147 BC00147 V=11.0  +MOVJ EC00147
SMOVC C00148 BC00148 V=11.0  +MOVJ EC00148
SMOVC C00149 BC00149 V=11.0  +MOVJ EC00149
ARCOF
SMOVL C00150 BC00150 V=400.0  +MOVJ EC00150
SMOVL C00151 BC00151 V=1000.0  +MOVJ EC00151
SFTOF3D
'Path W1580
SFTOF3D
SFTON3D P035
SMOVL C00152 BC00152 V=400.0  +MOVJ EC00152
SMOVL C00153 BC00153 V=100.0 PL=0  +MOVJ EC00153
SREFP 1 C00154 BC00154  +REFP EC00154
SREFP 2 C00155 BC00155  +REFP EC00155
MACRO1 MJ#(0) ARGF0
ARCON
SMOVC C00156 BC00156 V=11.0  +MOVJ EC00156
SMOVC C00157 BC00157 V=11.0  +MOVJ EC00157
SMOVC C00158 BC00158 V=11.0  +MOVJ EC00158
ARCOF
SMOVL C00159 BC00159 V=400.0  +MOVJ EC00159
SMOVL C00160 BC00160 V=1000.0  +MOVJ EC00160
SMOVL C00161 BC00161 V=1000.0  +MOVJ EC00161
SFTOF3D
MOVJ C00162 BC00162 VJ=100.00  +MOVJ EC00162 VJ=100.00
SFTOF
SFTON P035
'
MOVJ C00163 BC00163 VJ=50.00  +MOVJ EC00163 VJ=50.00
SMOVL C00164 BC00164 V=66.7  +MOVJ EC00164
SMOVL C00165 BC00165 V=66.7 PL=0  +MOVJ EC00165
MACRO1 MJ#(0) ARGF10
ARCON
SMOVC C00166 BC00166 V=10.0  +MOVJ EC00166
SMOVC C00167 BC00167 V=10.0  +MOVJ EC00167
SMOVC C00168 BC00168 V=10.0  +MOVJ EC00168
ARCOF
SMOVL C00169 BC00169 V=10.0  +MOVJ EC00169
SMOVL C00170 BC00170 V=66.7  +MOVJ EC00170
'Path W1106
SFTOF3D
SFTON3D P034
MOVJ C00171 BC00171 VJ=100.00  +MOVJ EC00171 VJ=100.00
SMOVL C00172 BC00172 V=400.0  +MOVJ EC00172
SMOVL C00173 BC00173 V=100.0 PL=0  +MOVJ EC00173
SREFP 1 C00174 BC00174  +REFP EC00174
SREFP 2 C00175 BC00175  +REFP EC00175
MACRO1 MJ#(0) ARGF0
ARCON
SMOVC C00176 BC00176 V=11.0  +MOVJ EC00176
SMOVC C00177 BC00177 V=11.0  +MOVJ EC00177
SMOVC C00178 BC00178 V=11.0  +MOVJ EC00178
ARCOF
SMOVL C00179 BC00179 V=400.0  +MOVJ EC00179
SFTOF3D
MOVJ C00180 BC00180 VJ=100.00  +MOVJ EC00180 VJ=100.00
'Path W1107
SFTOF3D
SFTON3D P034
MOVJ C00181 BC00181 VJ=100.00  +MOVJ EC00181 VJ=100.00
MOVJ C00182 BC00182 VJ=100.00  +MOVJ EC00182 VJ=100.00
SMOVL C00183 BC00183 V=400.0  +MOVJ EC00183
SMOVL C00184 BC00184 V=100.0 PL=0  +MOVJ EC00184
SREFP 1 C00185 BC00185  +REFP EC00185
SREFP 2 C00186 BC00186  +REFP EC00186
MACRO1 MJ#(0) ARGF0
ARCON
SMOVC C00187 BC00187 V=11.0  +MOVJ EC00187
SMOVC C00188 BC00188 V=11.0  +MOVJ EC00188
SMOVC C00189 BC00189 V=11.0  +MOVJ EC00189
ARCOF
SMOVL C00190 BC00190 V=400.0  +MOVJ EC00190
SFTOF3D
'Path W1108
SFTOF3D
SFTON3D P034
SMOVL C00191 BC00191 V=400.0  +MOVJ EC00191
SMOVL C00192 BC00192 V=100.0 PL=0  +MOVJ EC00192
SREFP 1 C00193 BC00193  +REFP EC00193
SREFP 2 C00194 BC00194  +REFP EC00194
MACRO1 MJ#(0) ARGF0
ARCON
SMOVC C00195 BC00195 V=11.0  +MOVJ EC00195
SMOVC C00196 BC00196 V=11.0  +MOVJ EC00196
SMOVC C00197 BC00197 V=11.0  +MOVJ EC00197
ARCOF
SMOVL C00198 BC00198 V=400.0  +MOVJ EC00198
SMOVL C00199 BC00199 V=1000.0  +MOVJ EC00199
SFTOF3D
'Path W1138
SFTOF3D
SFTON3D P033
MOVJ C00200 BC00200 VJ=100.00  +MOVJ EC00200 VJ=100.00
SMOVL C00201 BC00201 V=400.0  +MOVJ EC00201
SMOVL C00202 BC00202 V=100.0 PL=0  +MOVJ EC00202
SREFP 1 C00203 BC00203  +REFP EC00203
SREFP 2 C00204 BC00204  +REFP EC00204
MACRO1 MJ#(0) ARGF0
ARCON
SMOVC C00205 BC00205 V=11.0  +MOVJ EC00205
SMOVC C00206 BC00206 V=11.0  +MOVJ EC00206
SMOVC C00207 BC00207 V=11.0  +MOVJ EC00207
ARCOF
SMOVL C00208 BC00208 V=400.0  +MOVJ EC00208
SMOVL C00209 BC00209 V=1000.0  +MOVJ EC00209
SMOVL C00210 BC00210 V=1000.0  +MOVJ EC00210
SFTOF3D
'
'Path W1581
SFTOF3D
SFTON3D P033
SMOVL C00211 BC00211 V=100.0 PL=0  +MOVJ EC00211
SREFP 1 C00212 BC00212  +REFP EC00212
SREFP 2 C00213 BC00213  +REFP EC00213
MACRO1 MJ#(0) ARGF0
ARCON
SMOVC C00214 BC00214 V=11.0  +MOVJ EC00214
SMOVC C00215 BC00215 V=11.0  +MOVJ EC00215
SMOVC C00216 BC00216 V=11.0  +MOVJ EC00216
ARCOF
SMOVL C00217 BC00217 V=400.0  +MOVJ EC00217
SFTOF3D
MOVJ C00218 BC00218 VJ=100.00  +MOVJ EC00218 VJ=100.00
'Path W1582
SFTOF3D
SFTON3D P033
MOVJ C00219 BC00219 VJ=100.00  +MOVJ EC00219 VJ=100.00
MOVJ C00220 BC00220 VJ=100.00  +MOVJ EC00220 VJ=100.00
SMOVL C00221 BC00221 V=400.0  +MOVJ EC00221
SMOVL C00222 BC00222 V=100.0 PL=0  +MOVJ EC00222
SREFP 1 C00223 BC00223  +REFP EC00223
SREFP 2 C00224 BC00224  +REFP EC00224
MACRO1 MJ#(0) ARGF0
ARCON
SMOVC C00225 BC00225 V=11.0  +MOVJ EC00225
SMOVC C00226 BC00226 V=11.0  +MOVJ EC00226
SMOVC C00227 BC00227 V=11.0  +MOVJ EC00227
ARCOF
SMOVL C00228 BC00228 V=400.0  +MOVJ EC00228
SMOVL C00229 BC00229 V=1000.0  +MOVJ EC00229
SMOVL C00230 BC00230 V=66.7  +MOVJ EC00230
SFTOF3D
'Path W1583
SFTOF3D
SFTON3D P032
MOVJ C00231 BC00231 VJ=100.00  +MOVJ EC00231 VJ=100.00
SMOVL C00232 BC00232 V=400.0  +MOVJ EC00232
SMOVL C00233 BC00233 V=100.0 PL=0  +MOVJ EC00233
SREFP 1 C00234 BC00234  +REFP EC00234
SREFP 2 C00235 BC00235  +REFP EC00235
MACRO1 MJ#(0) ARGF0
ARCON
SMOVC C00236 BC00236 V=11.0  +MOVJ EC00236
SMOVC C00237 BC00237 V=11.0  +MOVJ EC00237
SMOVC C00238 BC00238 V=11.0  +MOVJ EC00238
ARCOF
SMOVL C00239 BC00239 V=400.0  +MOVJ EC00239
SMOVL C00240 BC00240 V=1000.0  +MOVJ EC00240
SFTOF3D
'Path W1584
SFTOF3D
SFTON3D P032
SMOVL C00241 BC00241 V=400.0  +MOVJ EC00241
SMOVL C00242 BC00242 V=100.0 PL=0  +MOVJ EC00242
SREFP 1 C00243 BC00243  +REFP EC00243
SREFP 2 C00244 BC00244  +REFP EC00244
MACRO1 MJ#(0) ARGF0
ARCON
SMOVC C00245 BC00245 V=11.0  +MOVJ EC00245
SMOVC C00246 BC00246 V=11.0  +MOVJ EC00246
SMOVC C00247 BC00247 V=11.0  +MOVJ EC00247
ARCOF
SMOVL C00248 BC00248 V=400.0  +MOVJ EC00248
SMOVL C00249 BC00249 V=1000.0  +MOVJ EC00249
SMOVL C00250 BC00250 V=1000.0  +MOVJ EC00250
SFTOF3D
MOVJ C00251 BC00251 VJ=100.00  +MOVJ EC00251 VJ=100.00
'
'Path W1109
SFTOF3D
SFTON3D P032
SMOVL C00252 BC00252 V=400.0  +MOVJ EC00252
SMOVL C00253 BC00253 V=100.0 PL=0  +MOVJ EC00253
SREFP 1 C00254 BC00254  +REFP EC00254
SREFP 2 C00255 BC00255  +REFP EC00255
MACRO1 MJ#(0) ARGF0
ARCON
SMOVC C00256 BC00256 V=11.0  +MOVJ EC00256
SMOVC C00257 BC00257 V=11.0  +MOVJ EC00257
SMOVC C00258 BC00258 V=11.0  +MOVJ EC00258
ARCOF
SMOVL C00259 BC00259 V=400.0  +MOVJ EC00259
SFTOF3D
MOVJ C00260 BC00260 VJ=100.00  +MOVJ EC00260 VJ=100.00
'Path W1110
SFTOF3D
SFTON3D P031
MOVJ C00261 BC00261 VJ=100.00  +MOVJ EC00261 VJ=100.00
SMOVL C00262 BC00262 V=400.0  +MOVJ EC00262
SMOVL C00263 BC00263 V=100.0 PL=0  +MOVJ EC00263
SREFP 1 C00264 BC00264  +REFP EC00264
SREFP 2 C00265 BC00265  +REFP EC00265
MACRO1 MJ#(0) ARGF0
ARCON
SMOVC C00266 BC00266 V=11.0  +MOVJ EC00266
SMOVC C00267 BC00267 V=11.0  +MOVJ EC00267
SMOVC C00268 BC00268 V=11.0  +MOVJ EC00268
ARCOF
SMOVL C00269 BC00269 V=400.0  +MOVJ EC00269
SMOVL C00270 BC00270 V=1000.0  +MOVJ EC00270
SFTOF3D
'Path W1111
SFTOF3D
SFTON3D P031
MOVJ C00271 BC00271 VJ=100.00  +MOVJ EC00271 VJ=100.00
SMOVL C00272 BC00272 V=400.0  +MOVJ EC00272
SMOVL C00273 BC00273 V=100.0 PL=0  +MOVJ EC00273
SREFP 1 C00274 BC00274  +REFP EC00274
SREFP 2 C00275 BC00275  +REFP EC00275
MACRO1 MJ#(0) ARGF0
ARCON
SMOVC C00276 BC00276 V=11.0  +MOVJ EC00276
SMOVC C00277 BC00277 V=11.0  +MOVJ EC00277
SMOVC C00278 BC00278 V=11.0  +MOVJ EC00278
ARCOF
SMOVL C00279 BC00279 V=400.0  +MOVJ EC00279
SMOVL C00280 BC00280 V=1000.0  +MOVJ EC00280
SFTOF3D
'Path W1139
SFTOF3D
SFTON3D P031
SMOVL C00281 BC00281 V=400.0  +MOVJ EC00281
SMOVL C00282 BC00282 V=100.0 PL=0  +MOVJ EC00282
SREFP 1 C00283 BC00283  +REFP EC00283
SREFP 2 C00284 BC00284  +REFP EC00284
MACRO1 MJ#(0) ARGF0
ARCON
SMOVC C00285 BC00285 V=11.0  +MOVJ EC00285
SMOVC C00286 BC00286 V=11.0  +MOVJ EC00286
SMOVC C00287 BC00287 V=11.0  +MOVJ EC00287
ARCOF
SMOVL C00288 BC00288 V=400.0  +MOVJ EC00288
SMOVL C00289 BC00289 V=1000.0  +MOVJ EC00289
SMOVL C00290 BC00290 V=1000.0  +MOVJ EC00290
SFTOF3D
MOVJ C00291 BC00291 VJ=100.00  +MOVJ EC00291 VJ=100.00
'
'Path W1585
SFTOF3D
SFTON3D P031
SMOVL C00292 BC00292 V=400.0  +MOVJ EC00292
SMOVL C00293 BC00293 V=100.0 PL=0  +MOVJ EC00293
SREFP 1 C00294 BC00294  +REFP EC00294
SREFP 2 C00295 BC00295  +REFP EC00295
MACRO1 MJ#(0) ARGF0
ARCON
SMOVC C00296 BC00296 V=11.0  +MOVJ EC00296
SMOVC C00297 BC00297 V=11.0  +MOVJ EC00297
SMOVC C00298 BC00298 V=11.0  +MOVJ EC00298
ARCOF
SMOVL C00299 BC00299 V=400.0  +MOVJ EC00299
SFTOF3D
'Path W1586
SFTOF3D
SFTON3D P031
SMOVL C00300 BC00300 V=400.0  +MOVJ EC00300
SMOVL C00301 BC00301 V=100.0 PL=0  +MOVJ EC00301
SREFP 1 C00302 BC00302  +REFP EC00302
SREFP 2 C00303 BC00303  +REFP EC00303
MACRO1 MJ#(0) ARGF0
ARCON
SMOVC C00304 BC00304 V=11.0  +MOVJ EC00304
SMOVC C00305 BC00305 V=11.0  +MOVJ EC00305
SMOVC C00306 BC00306 V=11.0  +MOVJ EC00306
ARCOF
SMOVL C00307 BC00307 V=400.0  +MOVJ EC00307
SMOVL C00308 BC00308 V=1000.0  +MOVJ EC00308
SFTOF3D
'Path W1587
SFTOF3D
SFTON3D P031
MOVJ C00309 BC00309 VJ=100.00  +MOVJ EC00309 VJ=100.00
SMOVL C00310 BC00310 V=400.0  +MOVJ EC00310
SMOVL C00311 BC00311 V=100.0 PL=0  +MOVJ EC00311
SREFP 1 C00312 BC00312  +REFP EC00312
SREFP 2 C00313 BC00313  +REFP EC00313
MACRO1 MJ#(0) ARGF0
ARCON
SMOVC C00314 BC00314 V=11.0  +MOVJ EC00314
SMOVC C00315 BC00315 V=11.0  +MOVJ EC00315
SMOVC C00316 BC00316 V=11.0  +MOVJ EC00316
ARCOF
SMOVL C00317 BC00317 V=400.0  +MOVJ EC00317
SMOVL C00318 BC00318 V=1000.0  +MOVJ EC00318
SFTOF3D
'OK
'OK
'OK
'OK
'OK
'Path W1588
SFTOF3D
SFTON3D P032
MOVJ C00319 BC00319 VJ=100.00  +MOVJ EC00319 VJ=100.00
SMOVL C00320 BC00320 V=400.0  +MOVJ EC00320
SMOVL C00321 BC00321 V=100.0 PL=0  +MOVJ EC00321
SREFP 1 C00322 BC00322  +REFP EC00322
SREFP 2 C00323 BC00323  +REFP EC00323
MACRO1 MJ#(0) ARGF0
ARCON
SMOVC C00324 BC00324 V=10.0  +MOVJ EC00324
SMOVC C00325 BC00325 V=10.0  +MOVJ EC00325
SMOVC C00326 BC00326 V=10.0  +MOVJ EC00326
ARCOF
SMOVL C00327 BC00327 V=400.0  +MOVJ EC00327
SMOVL C00328 BC00328 V=1000.0  +MOVJ EC00328
SMOVL C00329 BC00329 V=1000.0  +MOVJ EC00329
'Path W1112
SFTOF3D
SFTON3D P032
SMOVL C00330 BC00330 V=400.0  +MOVJ EC00330
SMOVL C00331 BC00331 V=100.0 PL=0  +MOVJ EC00331
SREFP 1 C00332 BC00332  +REFP EC00332
SREFP 2 C00333 BC00333  +REFP EC00333
MACRO1 MJ#(0) ARGF0
ARCON
SMOVC C00334 BC00334 V=10.0  +MOVJ EC00334
SMOVC C00335 BC00335 V=10.0  +MOVJ EC00335
SMOVC C00336 BC00336 V=10.0  +MOVJ EC00336
ARCOF
SMOVL C00337 BC00337 V=400.0  +MOVJ EC00337
SFTOF3D
MOVJ C00338 BC00338 VJ=100.00  +MOVJ EC00338 VJ=100.00
'Path W1113
SFTOF3D
SFTON3D P032
SMOVL C00339 BC00339 V=400.0  +MOVJ EC00339
SMOVL C00340 BC00340 V=100.0 PL=0  +MOVJ EC00340
SREFP 1 C00341 BC00341  +REFP EC00341
SREFP 2 C00342 BC00342  +REFP EC00342
MACRO1 MJ#(0) ARGF0
ARCON
SMOVC C00343 BC00343 V=10.0  +MOVJ EC00343
SMOVC C00344 BC00344 V=10.0  +MOVJ EC00344
SMOVC C00345 BC00345 V=10.0  +MOVJ EC00345
ARCOF
SMOVL C00346 BC00346 V=400.0  +MOVJ EC00346
SMOVL C00347 BC00347 V=1000.0  +MOVJ EC00347
SFTOF3D
'Path W1114
SFTOF3D
SFTON3D P033
SMOVL C00348 BC00348 V=400.0  +MOVJ EC00348
SMOVL C00349 BC00349 V=400.0  +MOVJ EC00349
SMOVL C00350 BC00350 V=100.0 PL=0  +MOVJ EC00350
SREFP 1 C00351 BC00351  +REFP EC00351
SREFP 2 C00352 BC00352  +REFP EC00352
MACRO1 MJ#(0) ARGF0
ARCON
SMOVC C00353 BC00353 V=10.0  +MOVJ EC00353
SMOVC C00354 BC00354 V=10.0  +MOVJ EC00354
SMOVC C00355 BC00355 V=10.0  +MOVJ EC00355
ARCOF
SMOVL C00356 BC00356 V=400.0  +MOVJ EC00356
SMOVL C00357 BC00357 V=1000.0  +MOVJ EC00357
SFTOF3D
'Path W1140
SFTOF3D
SFTON3D P033
SMOVL C00358 BC00358 V=400.0  +MOVJ EC00358
SMOVL C00359 BC00359 V=100.0 PL=0  +MOVJ EC00359
SREFP 1 C00360 BC00360  +REFP EC00360
SREFP 2 C00361 BC00361  +REFP EC00361
MACRO1 MJ#(0) ARGF0
ARCON
SMOVC C00362 BC00362 V=10.0  +MOVJ EC00362
SMOVC C00363 BC00363 V=10.0  +MOVJ EC00363
SMOVC C00364 BC00364 V=10.0  +MOVJ EC00364
ARCOF
SMOVL C00365 BC00365 V=400.0  +MOVJ EC00365
SMOVL C00366 BC00366 V=1000.0  +MOVJ EC00366
SMOVL C00367 BC00367 V=1000.0  +MOVJ EC00367
SFTOF3D
'
'Path W1589
SFTOF3D
SFTON3D P033
SMOVL C00368 BC00368 V=400.0  +MOVJ EC00368
SMOVL C00369 BC00369 V=100.0 PL=0  +MOVJ EC00369
SREFP 1 C00370 BC00370  +REFP EC00370
SREFP 2 C00371 BC00371  +REFP EC00371
MACRO1 MJ#(0) ARGF0
ARCON
SMOVC C00372 BC00372 V=10.0  +MOVJ EC00372
SMOVC C00373 BC00373 V=10.0  +MOVJ EC00373
SMOVC C00374 BC00374 V=10.0  +MOVJ EC00374
ARCOF
SMOVL C00375 BC00375 V=400.0  +MOVJ EC00375
SFTOF3D
MOVJ C00376 BC00376 VJ=100.00  +MOVJ EC00376 VJ=100.00
MOVJ C00377 BC00377 VJ=50.00  +MOVJ EC00377 VJ=50.00
MOVJ C00378 BC00378 VJ=50.00  +MOVJ EC00378 VJ=50.00
SFTOF
MOVJ C00379 BC00379 VJ=50.00  +MOVJ EC00379 VJ=50.00
END
